// TIA Portal V19 export
TYPE "FeedMachine_CIn"
// stored: Access Published
   STRUCT
      Manager : "FeedMachine_Manager";
      Bwd_ExtEnable : Bool := TRUE;
      Fwd_ExtEnable : Bool := TRUE;
      EnableManChangeVel : Bool := TRUE;   // Enable working of Manual velocity change Low to High
      ExternalAlarms : Bool := FALSE;
      VelocityOverride : Struct
         Enable : Bool := FALSE;
         Value : LReal := 100.0;   // %
      END_STRUCT;
   END_STRUCT;
END_TYPE
